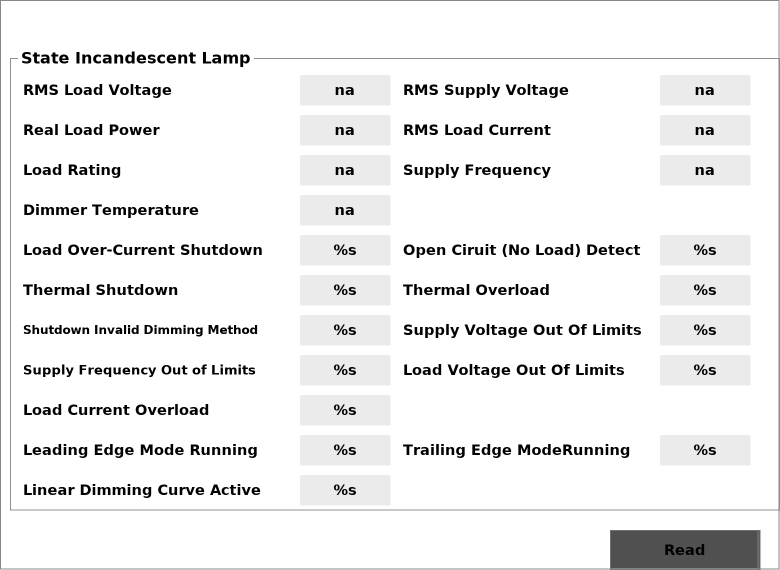
VISUALIZATION Visu_Part205Status  // 780x570
    Button (610,530 150x40), "Read"
        OnMouseClick: execute { DALI_Commissioning.fbPart205Incandescent.bReadStatus := TRUE; }
    GroupBox (10,50 770x460), "State Incandescent Lamp"
        Textfield (290,185 90x30), "%s", text variable: DALI_Commissioning.fbPart205Incandescent.sLoadOverCurrentShutdown
        Textfield (650,105 90x30), "%d Hz", text variable: DALI_Commissioning.fbPart205Incandescent.nSupplyFrequency
        Textfield (650,65 90x30), "%d %%", text variable: DALI_Commissioning.fbPart205Incandescent.nRMSLoadCurrent
        Textfield (650,25 90x30), "%d V", text variable: DALI_Commissioning.fbPart205Incandescent.nRMSSupplyVoltage
        Textfield (290,145 90x30), "%d °C", text variable: DALI_Commissioning.fbPart205Incandescent.nDimmerTemperature
        Textfield (290,105 90x30), "%2.1f mA", text variable: DALI_Commissioning.fbPart205Incandescent.fLoadRating
        Textfield (290,65 90x30), "%5.1f W", text variable: DALI_Commissioning.fbPart205Incandescent.fRealLoadPower
        Textfield (290,25 90x30), "%d V", text variable: DALI_Commissioning.fbPart205Incandescent.nRmsLoadVoltage
        Textfield (10,25 240x30), "RMS Load Voltage"
        Textfield (10,65 240x30), "Real Load Power", text variable: DALI_Commissioning.fbPart202Emergency.fFunctionTestDelayTimeVisu
        Textfield (10,145 240x30), "Dimmer Temperature"
        Textfield (10,105 240x30), "Load Rating"
        Textfield (10,185 240x30), "Load Over-Current Shutdown"
        Textfield (10,225 240x30), "Thermal Shutdown"
        Textfield (10,265 240x30), "Shutdown Invalid Dimming Method"
        Textfield (10,305 240x30), "Supply Frequency Out of Limits"
        Textfield (10,345 240x30), "Load Current Overload"
        Textfield (10,385 240x30), "Leading Edge Mode Running"
        Textfield (10,425 240x30), "Linear Dimming Curve Active"
        Textfield (290,265 90x30), "%s", text variable: DALI_Commissioning.fbPart205Incandescent.sInvalidDimmingMethod
        Textfield (290,305 90x30), "%s", text variable: DALI_Commissioning.fbPart205Incandescent.sSupplyFrequencyOutOfLimit
        Textfield (650,185 90x30), "%s", text variable: DALI_Commissioning.fbPart205Incandescent.sOpenCircuitDetection
        Textfield (650,225 90x30), "%s", text variable: DALI_Commissioning.fbPart205Incandescent.sThermalOverload
        Textfield (650,265 90x30), "%s", text variable: DALI_Commissioning.fbPart205Incandescent.sSupplyVoltageOutOfLimit
        Textfield (650,385 90x30), "%s", text variable: DALI_Commissioning.fbPart205Incandescent.sTrailingEdgeModeRunning
        Textfield (290,345 90x30), "%s", text variable: DALI_Commissioning.fbPart205Incandescent.sLoadCurrentOverload
        Textfield (290,385 90x30), "%s", text variable: DALI_Commissioning.fbPart205Incandescent.sLeadingEdgeModeRunning
        Textfield (290,425 90x30), "%s", text variable: DALI_Commissioning.fbPart205Incandescent.sLinearDimmingCurve
        Textfield (290,225 90x30), "%s", text variable: DALI_Commissioning.fbPart205Incandescent.sThermalShutdown
        Textfield (390,25 240x30), "RMS Supply Voltage"
        Textfield (390,65 240x30), "RMS Load Current"
        Textfield (390,105 240x30), "Supply Frequency"
        Textfield (390,185 240x30), "Open Ciruit (No Load) Detect"
        Textfield (390,225 240x30), "Thermal Overload"
        Textfield (390,265 240x30), "Supply Voltage Out Of Limits"
        Textfield (390,305 240x30), "Load Voltage Out Of Limits"
        Textfield (390,385 240x30), "Trailing Edge ModeRunning"
        Textfield (650,305 90x30), "%s", text variable: DALI_Commissioning.fbPart205Incandescent.sLoadVoltageOutOfLimit
        Textfield (290,25 90x30), "na", invisible if: not DALI_Commissioning.fbPart205Incandescent.bNoRmsLoadVoltage, input disabled if: true
        Textfield (290,65 90x30), "na", invisible if: not DALI_Commissioning.fbPart205Incandescent.bNoRealLoadPower, input disabled if: true
        Textfield (290,105 90x30), "na", invisible if: not DALI_Commissioning.fbPart205Incandescent.bNoLoadRating, input disabled if: true
        Textfield (290,145 90x30), "na", invisible if: not DALI_Commissioning.fbPart205Incandescent.bNoDimmerTemperature, input disabled if: true
        Textfield (650,25 90x30), "na", invisible if: not DALI_Commissioning.fbPart205Incandescent.bNoRMSSupplyVoltage, input disabled if: true
        Textfield (650,65 90x30), "na", invisible if: not DALI_Commissioning.fbPart205Incandescent.bNoRMSLoadCurrent, input disabled if: true
        Textfield (650,105 90x30), "na", invisible if: not DALI_Commissioning.fbPart205Incandescent.bNoSupplyFrequency, input disabled if: true
END_VISUALIZATION

(* stored: Version 1.1.0.1, ProductVersion 3.1.4024.12
   Visu Visu_Part205Status: Id {6ffa27e1-9d9c-441b-a825-10e3cc532ec6} *)
